FUNCTION_BLOCK CardboardCornerGuardEx
VAR_IN_OUT //controls
	execute : BOOL;
	stop : BOOL;
	
	manualStep : BOOL;
	manualSuction : BOOL;
END_VAR
VAR_IN_OUT
	benderLeft : FoldingMachine;
	
	robotLeft, robotRight : RobotA22;
	
	skidLeft, skidRight : SkidMagazine;
	magazineLeft, magazineRight : SkidMagazine;
	
	wrapper : WrapMachine;
	
	horizontalDriveLeft, horizontalDriveRight : ServoNC;
	verticalDriveLeft, verticalDriveRight : ClearLinkMC;
	pistonBottom : SimplePiston;
	
	suctionTopLeft : ARRAY[*(*1..3*)] OF SuctionPad;
	suctionTopRight : ARRAY[*(*1..3*)] OF SuctionPad;
	suctionBottomLeft : ARRAY[*(*1..3*)] OF SuctionPad; 
	suctionBottomRight : ARRAY[*(*1..3*)] OF SuctionPad;
END_VAR
VAR_OUTPUT
	generalError : BOOL;
	failLeft, failRight : BOOL;
END_VAR
VAR //for testing only
	latchLeft, latchRight : BOOL; //prevents sliders from overshooting the inner limit sensor
	
	suctionEnableTopLeft : BOOL;
	suctionEnableTopRight : BOOL;
	suctionEnableBottomLeft : BOOL;
	suctionEnableBottomRight : BOOL;
	
	ready : BOOL;
	done : BOOL;
END_VAR
VAR	
	step : (IDLE, LOAD_CORNERS, LOAD_FLATS, PUSH, TARGET_WRAP_POSITION, WRAP_AND_RELEASE, COMPLETE := 1050);
	iPair : INT;
	
	masterLoadStep : INT;
	loadSet : INT;
	loadStepLeft, loadStepRight : INT;
	cornerSetLeft, cornerSetRight : INT;
	
	iWrap : INT;
	wrapPoints : INT;
	wrapRotations : INT;
	masterLength : INT;
	
	releaseDelayTimer : TON;
END_VAR
VAR //local types
	topLeftFoldsArr, topRightFoldsArr, bottomLeftFoldsArr, bottomRightFoldsArr : ARRAY[0..GVL.maxPairs] OF INT;
	materialsArr : ARRAY[0..GVL.maxPairs] OF PositionMaterials := [
		(
			position := 0,
			top := 'CAR20M',
			left := 'CAR20S',
			right := 'CAR20S',
			bottom := 'CAR20L',
			topLeft := 'CAR28M',
			topRight := 'CAR28S',
			bottomLeft := 'CAR28S',
			bottomRight := 'CAR28L',
			wrapPoints := 1,
			wrapRotations := 4
		),
		(
			position := 0,
			topLeft := 'COR48',
			topRight := 'COR48',
			bottomLeft := 'COR48',
			bottomRight := 'COR48'
		)];
	
	demoHeight : REAL := 600; //600mm, 60cm
	
	insertionLeft, insertionRight : Insertion;
	innerLoadedMaterials, outerLoadedMaterials : ARRAY[Surface.TOP..Surface.BOTTOM_RIGHT] OF STRING;
	//inner: cardboard by default
	//outer: corner guard by default
END_VAR
VAR CONSTANT
	sectionID : SectionEnum := SectionEnum.CARDBOARD_CORNERGUARD;
	releaseDelay : TIME := T#2000MS;
END_VAR
VAR
	//AOIs encapsulate functionality and reduce the number of module variables
	aoiLoadCornerGuardLeft, aoiLoadCornerGuardRight : AOI_LoadCornerGuard;
	aoiLoadFlatCardboardLeft, aoiLoadFlatCardboardRight : AOI_LoadFlatCardboard;
END_VAR

callLocalModules();

IF stop THEN //may need to turn off suction
	insertionLeft.stop();
	insertionRight.stop();
	pistonBottom.stop();
	
	robotLeft.clearCommand();
	robotRight.clearCommand();
	RETURN;
END_IF

IF NOT (insertionLeft.homingComplete AND insertionRight.homingComplete) THEN
	insertionLeft.homingSequence();
	insertionRight.homingSequence();
	pistonBottom.retract();
END_IF

CASE step OF
	IDLE:
		IF execute THEN
			execute := FALSE;
			step := LOAD_CORNERS;
		END_IF
	
	LOAD_CORNERS:
		IF load(pairIndex := iPair) THEN
			IF manualStep AND_THEN NOT execute THEN
				RETURN;
			END_IF
		
			step := LOAD_FLATS;
		END_IF

	LOAD_FLATS:
		IF loadFlats(pair := materialsArr[iPair]) THEN
			IF manualStep AND_THEN NOT execute THEN
				RETURN;
			END_IF
			
			step := PUSH;
		END_IF
		
	PUSH:
		IF
			NOT insertionLeft.align(1000-demoHeight) OR
			NOT insertionRight.align(1000-demoHeight)
		THEN
			RETURN;
		END_IF
		
		insertionLeft.press();
		insertionRight.press();
		pistonBottom.extend();
		
		IF pistonBottom.extended AND insertionLeft.contact AND insertionRight.contact THEN
			step := TARGET_WRAP_POSITION;
		END_IF
		
	TARGET_WRAP_POSITION:		
		IF iWrap >= wrapPoints THEN
			step := COMPLETE;
			RETURN;
		END_IF
		
		//loadNextPair := materialsArr[iPair].position = materialsArr[iPair + 1].position;	
		
		IF materialsArr[iPair].position = materialsArr[iPair + 1].position THEN
			masterLength := MAX( GetPairMasterLength(materialsArr[iPair]), GetPairMasterLength(materialsArr[iPair + 1]) );
			wrapPoints := MAX( materialsArr[iPair].wrapPoints, materialsArr[iPair + 1].wrapPoints );
			wrapRotations := MAX( materialsArr[iPair].wrapRotations, materialsArr[iPair + 1].wrapRotations );
		ELSE
			masterLength := GetPairMasterLength(materialsArr[iPair]);
			wrapPoints := materialsArr[iPair].wrapPoints;
			wrapRotations := materialsArr[iPair].wrapRotations;
		END_IF
		
		(*
		directionCheckAndSet(
			wrapConveyorPos,
			(currentPair.position - masterLength/2) + (masterLength/(currentPair.wrapPoints + 1) * (iWrap + 1)));
		*)
		step := WRAP_AND_RELEASE;
		
	WRAP_AND_RELEASE:
		releaseDelayTimer(IN:= , PT:= releaseDelay, Q=> , ET=> );
		
		IF wrapper.ready THEN
			wrapper.wrap(wrapRotations);
			releaseDelayTimer.IN := TRUE;
		END_IF
		
		IF releaseDelayTimer.Q THEN
			SetSuctions(suctions := suctionTopLeft, state := FALSE);
			SetSuctions(suctions := suctionTopRight, state := FALSE);
			SetSuctions(suctions := suctionBottomLeft, state := FALSE);
			SetSuctions(suctions := suctionBottomRight, state := FALSE);
			
			insertionLeft.align(0);
			insertionRight.align(0);
			insertionLeft.release();
			insertionRight.release();
			
			pistonBottom.retract();
		END_IF
		
		IF wrapper.done AND insertionLeft.home AND insertionRight.home AND pistonBottom.retracted THEN
			releaseDelayTimer.IN := FALSE;
			step := WRAP_AND_RELEASE;
		END_IF
	
	COMPLETE:
		iPair := (iPair + 1) MOD GVL.maxPairs;
		iWrap := wrapPoints := wrapRotations := 0;
		step := IDLE;
		
END_CASE

ACTION blocks:
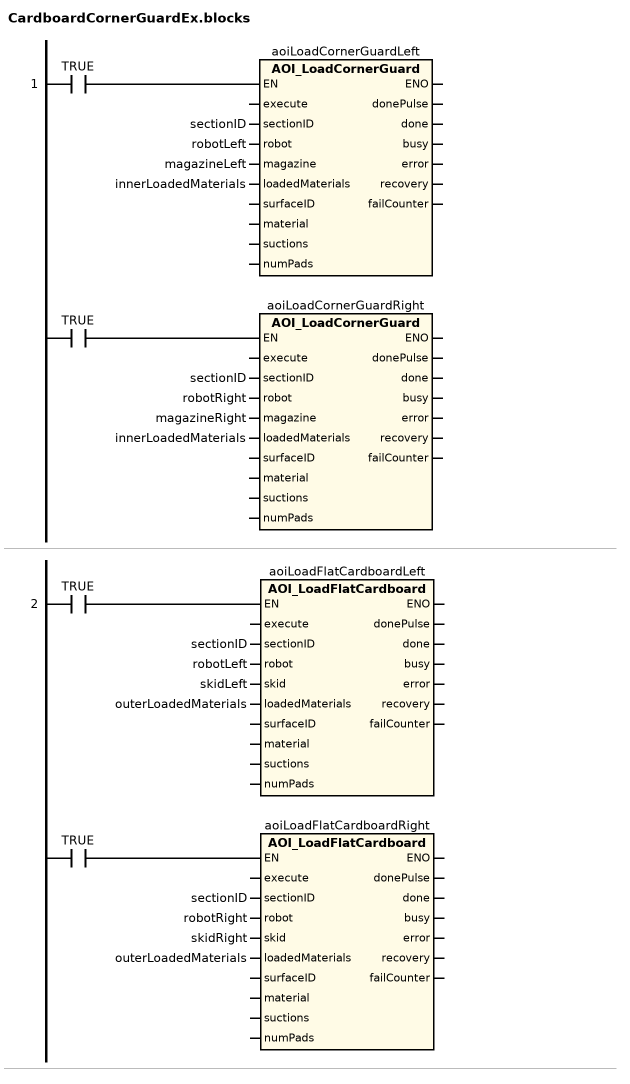
// NETWORK 1
aoiLoadCornerGuardLeft(
    sectionID := sectionID,
    robot := robotLeft,
    magazine := magazineLeft,
    loadedMaterials := innerLoadedMaterials); // AOI_LoadCornerGuard
aoiLoadCornerGuardRight(
    sectionID := sectionID,
    robot := robotRight,
    magazine := magazineRight,
    loadedMaterials := innerLoadedMaterials); // AOI_LoadCornerGuard

// NETWORK 2
aoiLoadFlatCardboardLeft(
    sectionID := sectionID,
    robot := robotLeft,
    skid := skidLeft,
    loadedMaterials := outerLoadedMaterials); // AOI_LoadFlatCardboard
aoiLoadFlatCardboardRight(
    sectionID := sectionID,
    robot := robotRight,
    skid := skidRight,
    loadedMaterials := outerLoadedMaterials); // AOI_LoadFlatCardboard
END_ACTION

ACTION callLocalModules:
{warning disable C0371}
insertionLeft(
	enable:= TRUE, 
	slider:= verticalDriveLeft, 
	screw:= horizontalDriveLeft, 
	contact=> , 
	softContact=> , 
	busy=> , 
	error=> , 
	home=> , 
	homingComplete=> , 
	sliderPos=> );
	
insertionRight(
	enable:= TRUE, 
	slider:= verticalDriveRight, 
	screw:= horizontalDriveRight, 
	contact=> , 
	softContact=> , 
	busy=> , 
	error=> , 
	home=> , 
	homingComplete=> , 
	sliderPos=> );
END_ACTION

METHOD PROTECTED leftCornerSequence : BOOL
VAR_IN_OUT
	robot : RobotA22;
	skid : SkidMagazine;
	suctions : POINTER TO SuctionPad; //ARRAY[*] OF SuctionPad;
	loadStep : INT;
END_VAR
VAR_INPUT
	surfaceID : Surface;
	material : STRING;
	foldPos0 : INT;
	foldPos1 : INT;
END_VAR
VAR_OUTPUT
	error : BOOL;
END_VAR
VAR
	column : INT;
END_VAR
VAR CONSTANT
	suctionDistance : INT := 10;
END_VAR
{warning disable C0371}
IF material = '' THEN
	leftCornerSequence := TRUE;
	RETURN;
END_IF

benderLeft.setFoldingPositions(foldPos0, foldPos1);

CASE loadStep OF
	0:
		robot.clearCommand();
		IF robot.Ready AND overhead = '' THEN
			loadStep := 10;
		END_IF
		
	10: //skid to bender
		IF NOT skid.findSlot(materialID:= material, index=> column) THEN
			error := TRUE;
			RETURN;
		END_IF
		
		(*
		IF robot.eoatDistance < suctionDistance THEN
			robot.HoldMaterial := skid.getSlot(i := column);
		END_IF
		*)
		
		IF robot.Done THEN
			loadStep := 20;
			RETURN;
		END_IF
		
		robot.setGroup(group := 1, value := A22.TRANSFER_TO_BENDER);
		robot.setGroup(group := 2, value := foldPos0);
		robot.setGroup(group := 3, value := foldPos1);
		
	20: //bend
		//IF benderLeft.done THEN
			loadStep := 30;
		//END_IF
		
	30: //bender to overhead or left insertion
		IF wrapper.trayOccupied AND wrapper.Overhead = '' AND robot.HoldMaterial <> '' THEN
			wrapper.Overhead := robot.HoldMaterial;
			robot.HoldMaterial := '';
		END_IF
	
		IF robot.Done THEN
			loadStep := COMPLETE;
			RETURN;
		END_IF
		
		CASE surfaceID OF
			Surface.TOP_RIGHT:		robot.setGroup(group := 1, value := A22.TRANSFER_TO_OVERHEAD);
			Surface.BOTTOM_RIGHT:	robot.setGroup(group := 1, value := A22.TRANSFER_TO_OVERHEAD);
			Surface.TOP_LEFT:		robot.setGroup(group := 1, value := A22.LOAD_BENDER_TO_UPPER_CORNER);
			Surface.BOTTOM_LEFT:	robot.setGroup(group := 1, value := A22.LOAD_BENDER_TO_LOWER_CORNER);
		END_CASE
		robot.setGroup(group := 2, value := 0);
		robot.setGroup(group := 3, value := 0);
	
	COMPLETE:
		CASE surfaceID OF
			Surface.TOP_LEFT:		suctionTopLeft[1].enable := suctionTopLeft[3].enable := TRUE;
			Surface.BOTTOM_LEFT:	suctionBottomLeft[1].enable := suctionBottomLeft[3].enable := TRUE;
		END_CASE
		
		leftCornerSequence := TRUE;
		
END_CASE
END_METHOD

METHOD PROTECTED load : BOOL
VAR_INPUT
	pairIndex : INT;
END_VAR
VAR
	pair : REFERENCE TO PositionMaterials REF= materialsArr[pairIndex];
	nextPair : REFERENCE TO PositionMaterials;
END_VAR
(*
unlike other sections, the load() function for cardboard + corner guard only loads the corners
to load flat cardboards, use the function loadFlats()
*)
{warning disable C0371}

IF robotLeft.error OR robotRight.error THEN
	RETURN;
ELSIF NOT (robotLeft.reserve(sectionID) AND robotRight.reserve(sectionID)) THEN //both robots must be reserved first
	RETURN;
END_IF

IF pairIndex + 1 < GVL.maxPairs THEN
	nextPair REF= materialsArr[pairIndex + 1];
END_IF

CASE masterLoadStep OF
	0: //next pair (which is to be placed over this pair) has the same position as this pair
		IF pairIndex + 1 >= GVL.maxPairs THEN //no next pair
			masterLoadStep := 10;
		ELSIF pair.position < nextPair.position THEN
			masterLoadStep := 10;
		ELSIF MatchesMaterialType(pair:= nextPair, materialType:= 'CAR') AND_THEN loadCornerCardboards(pairIndex:= pairIndex + 1) THEN
			masterLoadStep := 10;
		ELSIF MatchesMaterialType(pair:= nextPair, materialType:= 'COR') AND_THEN loadCornerGuards(pairIndex:= pairIndex + 1) THEN
			masterLoadStep := 10;
		END_IF
		
	10:
		IF
			MatchesMaterialType(pair:= pair, materialType:= 'CAR') AND_THEN loadCornerCardboardsEx(pairIndex:= iPair) OR_ELSE
			MatchesMaterialType(pair:= pair, materialType:= 'COR') AND_THEN loadCornerGuards(pairIndex:= iPair)
		THEN //is cardboard
			masterLoadStep := COMPLETE;
		END_IF
	
	COMPLETE:
		robotLeft.release(sectionID);
		robotRight.release(sectionID);
		
		masterLoadStep := 0;
		load := TRUE;
	
END_CASE
END_METHOD

METHOD PROTECTED loadCornerCardboards : BOOL
VAR_INPUT
	pairIndex : INT;
END_VAR
VAR
	leftSuctionArr, rightSuctionArr : POINTER TO SuctionPad;
	leftNextSet, rightNextSet : INT;
	leftMaterial, rightMaterial : STRING;
	leftFold, rightFold : INT;
	
	pair : REFERENCE TO PositionMaterials REF= materialsArr[pairIndex];
	topLeftFold : INT := topLeftFoldsArr[pairIndex];
	topRightFold : INT := topRightFoldsArr[pairIndex];
	bottomLeftFold : INT := bottomLeftFoldsArr[pairIndex];
	bottomRightFold : INT := bottomRightFoldsArr[pairIndex];
END_VAR
{warning disable C0371}
CASE cornerSetLeft OF
	0:
		leftNextSet := Surface.TOP_RIGHT;
		cornerSetLeft := 0;
		
	Surface.TOP_RIGHT: 
		leftNextSet := Surface.TOP_LEFT;
		leftSuctionArr := suctionTopRight;
		leftMaterial := pair.topRight;
		leftFold := topRightFold;
		
	Surface.TOP_LEFT: 
		leftNextSet := Surface.BOTTOM_RIGHT;
		leftSuctionArr := suctionTopLeft;
		leftMaterial := pair.topLeft;
		leftFold := topLeftFold;
		
	Surface.BOTTOM_RIGHT:
		leftNextSet := Surface.BOTTOM_LEFT;
		leftSuctionArr := suctionBottomRight;
		leftMaterial := pair.bottomRight;
		leftFold := bottomRightFold;
		
	Surface.BOTTOM_LEFT: 
		leftNextSet := COMPLETE;
		leftSuctionArr := suctionBottomLeft;
		leftMaterial := pair.bottomLeft;
		leftFold := bottomLeftFold;
END_CASE
IF
	(cornerSetLeft = 0 OR cornerSetLeft = COMPLETE) OR_ELSE
	leftCornerSequence(
		robot:= robotLeft, 
		skid:= skidLeft, 
		suctions := leftSuctionArr,
		loadStep:= loadStepLeft, 
		surfaceID:= cornerSetLeft,
		material:= pair.topRight, 
		foldPos0:= topRightFold, 
		foldPos1:= 0, 
		error=> )
THEN
	cornerSetLeft := leftNextSet;
	loadStepLeft := 0;
END_IF


CASE cornerSetRight OF
	0:
		cornerSetRight := Surface.TOP_RIGHT;
		rightSuctionArr := suctionTopRight;
		
	Surface.TOP_RIGHT:		
		rightNextSet := Surface.BOTTOM_RIGHT;
		rightSuctionArr := suctionTopRight;
		rightMaterial := pair.topRight;
		rightFold := topRightFold;
		
	Surface.BOTTOM_RIGHT: 
		rightNextSet := COMPLETE;
		rightSuctionArr := suctionBottomRight;
		rightMaterial := pair.bottomRight;
		rightFold := bottomRightFold;		
END_CASE
IF
	(cornerSetRight = 0 OR cornerSetRight = COMPLETE) OR_ELSE
	rightCornerSequence(
		robot:= robotRight, 
		skid:= skidRight, 
		suctions := rightSuctionArr,
		loadStep:= loadStepRight, 
		material:= pair.topRight, 
		surfaceID:= cornerSetRight,
		foldPos0:= pair.topRightFold, 
		foldPos1:= 0, 
		error=> )
THEN
	cornerSetRight := rightNextSet;
	loadStepRight := 0;
END_IF



IF cornerSetLeft = COMPLETE AND cornerSetRight = COMPLETE THEN
	loadCornerCardboards := TRUE;
	
	loadStepLeft := loadStepRight := 0;
	cornerSetLeft := cornerSetRight := 0;
END_IF
END_METHOD

METHOD PROTECTED loadCornerCardboardsEx : BOOL
VAR_INPUT
	pairIndex : INT;
END_VAR
VAR
	suctionsArrLeft, suctionsArrRight : POINTER TO SuctionPad;
	nextSetLeft, nextSetRight : INT;

	pair : REFERENCE TO PositionMaterials REF= materialsArr[pairIndex];
	topLeftFold : INT := topLeftFoldsArr[pairIndex];
	topRightFold : INT := topRightFoldsArr[pairIndex];
	bottomLeftFold : INT := bottomLeftFoldsArr[pairIndex];
	bottomRightFold : INT := bottomRightFoldsArr[pairIndex];
END_VAR
{warning disable C0371}
CASE cornerSetLeft OF
	0:
		cornerSetLeft := Surface.TOP_RIGHT;
		loadStepLeft := 0;
		
	Surface.TOP_RIGHT: 
		IF
			leftCornerSequence(
				robot:= robotLeft, 
				skid:= skidLeft, 
				suctions := suctionTopRight,
				loadStep:= loadStepLeft, 
				surfaceID:= Surface.TOP_RIGHT,
				material:= pair.topRight, 
				foldPos0:= topRightFold, 
				foldPos1:= 0, 
				error=> )
		THEN
			cornerSetLeft := Surface.TOP_LEFT;
			loadStepLeft := 0;
		END_IF
		
	Surface.TOP_LEFT: 
		IF
			leftCornerSequence(
				robot:= robotLeft, 
				skid:= skidLeft, 
				suctions := suctionTopLeft,
				loadStep:= loadStepLeft, 
				surfaceID:= Surface.TOP_LEFT,
				material:= pair.topLeft, 
				foldPos0:= topLeftFold, 
				foldPos1:= 0, 
				error=> )
		THEN
			cornerSetLeft := Surface.BOTTOM_RIGHT;
			loadStepLeft := 0;
		END_IF
		
	Surface.BOTTOM_RIGHT: 
		IF
			leftCornerSequence(
				robot:= robotLeft, 
				skid:= skidLeft, 
				suctions := suctionBottomRight,
				loadStep:= loadStepLeft, 
				surfaceID:= Surface.BOTTOM_RIGHT,
				material:= pair.bottomRight, 
				foldPos0:= bottomRightFold, 
				foldPos1:= 0, 
				error=> )
		THEN
			cornerSetLeft := Surface.BOTTOM_LEFT;
			loadStepLeft := 0;
		END_IF
		
	Surface.BOTTOM_LEFT: 
		IF
			leftCornerSequence(
				robot:= robotLeft, 
				skid:= skidLeft, 
				suctions := suctionBottomLeft,
				loadStep:= loadStepLeft, 
				surfaceID:= Surface.BOTTOM_LEFT,
				material:= pair.bottomLeft, 
				foldPos0:= bottomLeftFold, 
				foldPos1:= 0, 
				error=> )
		THEN
			cornerSetLeft := COMPLETE;
			loadStepLeft := 0;
		END_IF
END_CASE

//------------------------------------------------------------
CASE cornerSetRight OF
	0:
		cornerSetRight := Surface.TOP_RIGHT;
		loadStepRight := 0;
		
	Surface.TOP_RIGHT: 
		IF
			rightCornerSequence(
				robot:= robotRight, 
				skid:= skidRight, 
				suctions := suctionTopRight,
				loadStep:= loadStepRight, 
				surfaceID:= Surface.TOP_RIGHT,
				material:= pair.topRight, 
				foldPos0:= topRightFold, 
				foldPos1:= 0, 
				error=> )
		THEN
			cornerSetRight := Surface.BOTTOM_RIGHT;
			loadStepRight := 0;
		END_IF
		
	Surface.BOTTOM_RIGHT: 
		IF
			rightCornerSequence(
				robot:= robotRight, 
				skid:= skidRight, 
				suctions := suctionBottomRight,
				loadStep:= loadStepRight, 
				surfaceID:= Surface.BOTTOM_RIGHT,
				material:= pair.bottomRight, 
				foldPos0:= bottomRightFold, 
				foldPos1:= 0, 
				error=> )
		THEN
			cornerSetRight := Surface.BOTTOM_RIGHT;
			loadStepRight := 0;
		END_IF
		
		cornerSetRight := COMPLETE;			
		loadStepRight := COMPLETE;
		
END_CASE

//------------------------------------------------------------
IF cornerSetLeft = COMPLETE AND cornerSetRight = COMPLETE THEN
	loadCornerCardboardsEx := TRUE;
	
	loadStepLeft := loadStepRight := 0;
	cornerSetLeft := cornerSetRight := 0;
END_IF
END_METHOD

METHOD PROTECTED loadCornerGuards : BOOL
VAR_INPUT
	pairIndex : INT;
END_VAR
VAR_OUTPUT
	fail : BOOL;
END_VAR
VAR
	pair : REFERENCE TO PositionMaterials REF= materialsArr[pairIndex];
END_VAR
{warning disable C0371}
CASE loadSet OF
	0: //upper corners
		IF 
			loadGuardSequence(
				robot:= robotLeft, 
				magazine:= magazineLeft, 
				suctions:= suctionTopLeft,
				loadStep:= loadStepLeft, 
				surfaceID:= Surface.TOP_LEFT, 
				material:= pair.topLeft, 
				error=> failLeft)
			AND
			loadGuardSequence(
				robot:= robotRight, 
				magazine:= magazineLeft,
				suctions:= suctionTopRight,
				loadStep:= loadStepRight, 
				surfaceID:= Surface.TOP_RIGHT, 
				material:= pair.topRight, 
				error=> failRight)
		THEN
			loadStepLeft := loadStepRight := 0;
			loadSet := 10;
		END_IF
		
	10: //lower corners
		IF 
			loadGuardSequence(
				robot:= robotLeft, 
				magazine:= skidLeft, 
				suctions:= suctionTopLeft,
				loadStep:= loadStepLeft, 
				surfaceID:= Surface.BOTTOM_LEFT, 
				material:= pair.bottomLeft, 
				error=> failLeft)
			AND
			loadGuardSequence(
				robot:= robotRight, 
				magazine:= skidRight,
				suctions:= suctionTopRight,
				loadStep:= loadStepRight, 
				surfaceID:= Surface.BOTTOM_RIGHT, 
				material:= pair.bottomRight, 
				error=> failRight)
		THEN
			loadStepLeft := loadStepRight := 0;
			loadSet := COMPLETE;
		END_IF
	
	COMPLETE:
		loadStepLeft := loadStepRight := 0;
		loadSet := 0;
		
		loadCornerGuards := TRUE;
END_CASE

fail := failLeft OR failRight;
END_METHOD

METHOD PROTECTED loadFlats : BOOL
VAR_INPUT
	pair : REFERENCE TO PositionMaterials;
END_VAR
VAR_OUTPUT
	error : BOOL;
END_VAR
{warning disable C0371}
CASE loadSet OF
	0: //top and bottom
		IF 
			loadFlatSequence(
				robot:= robotLeft, 
				skid:= skidLeft, 
				loadStep:= loadStepLeft, 
				surfaceID:= Surface.TOP, 
				material:= pair.top, 
				fail=> )
			AND
			loadFlatSequence(
				robot:= robotRight, 
				skid:= skidRight, 
				loadStep:= loadStepRight, 
				surfaceID:= Surface.BOTTOM, 
				material:= pair.bottom, 
				fail=> )
		THEN
			loadStepLeft := loadStepRight := 0;
			loadSet := 10;
		END_IF
		
	10: //sides
		IF 
			loadFlatSequence(
				robot:= robotLeft, 
				skid:= skidLeft, 
				loadStep:= loadStepLeft, 
				surfaceID:= Surface.LEFT, 
				material:= pair.left, 
				fail=> )
			AND
			loadFlatSequence(
				robot:= robotRight, 
				skid:= skidRight, 
				loadStep:= loadStepRight, 
				surfaceID:= Surface.RIGHT, 
				material:= pair.right, 
				fail=> )
		THEN
			loadStepLeft := loadStepRight := 0;
			loadSet := COMPLETE;
		END_IF
	
	COMPLETE:
		loadStepLeft := loadStepRight := 0;
		loadSet := 0;
		
		loadFlats := TRUE;
END_CASE
END_METHOD

METHOD loadFlatSequence : BOOL
VAR_IN_OUT
	robot : RobotA22;
	skid : SkidMagazine;
	loadStep : INT;
END_VAR
VAR_INPUT
	surfaceID : Surface;
	material : STRING;
END_VAR
VAR_OUTPUT
	fail : BOOL;
END_VAR
VAR
	task : INT;
	slot : INT;
END_VAR
IF material = '' THEN
	loadFlatSequence := TRUE;
	RETURN;
END_IF

CASE loadStep OF
	0:
		robot.clearCommand();
		IF robot.Ready THEN
			step := 10;
		END_IF
		
	10: //storage to gripper
		IF NOT skid.findSlot(materialID := material, index => slot) THEN
			fail := TRUE;
			RETURN;
		END_IF
		
		IF robot.Done THEN
			loadStep := COMPLETE;
			RETURN;
		END_IF
		
		CASE surfaceID OF
			Surface.TOP: 					task := A22.LOAD_CARDBOARD_TOP;
			Surface.LEFT, Surface.RIGHT: 	task := A22.LOAD_CARDBOARD_SIDE;
			Surface.BOTTOM: 				task := A22.LOAD_CARDBOARD_BOTTOM;
		END_CASE
		
		robot.setGroup(group := 1, value := task);
		robot.setGroup(group := 2, value := slot);
		
	20: //gripper to insertion
		
	COMPLETE:
		loadFlatSequence := TRUE;
	
END_CASE
END_METHOD

METHOD loadGuardSequence : BOOL
VAR_IN_OUT
	robot : RobotA22;
	magazine : SkidMagazine;
	suctions : ARRAY[*] OF SuctionPad;
	loadStep : INT;
END_VAR
VAR_INPUT
	surfaceID : Surface;
	material : STRING;
END_VAR
VAR_OUTPUT
	error : BOOL;
END_VAR
VAR
	task : INT;
	slot : INT;
END_VAR
IF material = '' THEN
	loadGuardSequence := TRUE;
	RETURN;
END_IF

CASE loadStep OF
	0:
		IF NOT magazine.findSlot(materialID := material, index => slot) THEN //load from staging table
			error := TRUE;
			RETURN;
		END_IF
		
		IF robot.Done THEN
			loadStep := COMPLETE;
			RETURN;
		END_IF
		
		CASE surfaceID OF
			Surface.TOP_LEFT, Surface.TOP_RIGHT: 		task := A22.LOAD_CORNER_GUARD_UPPER;
			Surface.BOTTOM_LEFT, Surface.BOTTOM_RIGHT:	task := A22.LOAD_CORNER_GUARD_LOWER;
		END_CASE
		
		robot.setGroup(group := 1, value := task);
		robot.setGroup(group := 2, value := slot);
		
	COMPLETE:
		suctions[2].enable := TRUE;
		loadGuardSequence := TRUE;
END_CASE
END_METHOD

METHOD PROTECTED loadLeftCornerCardboards : BOOL
VAR_INPUT
	pair : REFERENCE TO PositionMaterials;
END_VAR
VAR
	suctionsArrLeft, suctionsArrRight : POINTER TO SuctionPad;
	nextSetLeft, nextSetRight : INT;
END_VAR
{warning disable C0371}
CASE cornerSetLeft OF
	0:
		cornerSetLeft := Surface.TOP_RIGHT;
		loadStepLeft := 0;
		
	Surface.TOP_RIGHT: 
		IF
			leftCornerSequence(
				robot:= robotLeft, 
				skid:= skidLeft, 
				suctions := suctionTopRight,
				loadStep:= loadStepLeft, 
				surfaceID:= Surface.TOP_RIGHT,
				material:= pair.topRight, 
				foldPos0:= pair.topRightFold, 
				foldPos1:= 0, 
				error=> )
		THEN
			cornerSetLeft := Surface.TOP_LEFT;
			loadStepLeft := 0;
		END_IF
		
	Surface.TOP_LEFT: 
		IF
			leftCornerSequence(
				robot:= robotLeft, 
				skid:= skidLeft, 
				suctions := suctionTopLeft,
				loadStep:= loadStepLeft, 
				surfaceID:= Surface.TOP_LEFT,
				material:= pair.topLeft, 
				foldPos0:= pair.topLeftFold, 
				foldPos1:= 0, 
				error=> )
		THEN
			cornerSetLeft := Surface.BOTTOM_RIGHT;
			loadStepLeft := 0;
		END_IF
		
	Surface.BOTTOM_RIGHT: 
		IF
			leftCornerSequence(
				robot:= robotLeft, 
				skid:= skidLeft, 
				suctions := suctionBottomRight,
				loadStep:= loadStepLeft, 
				surfaceID:= Surface.BOTTOM_RIGHT,
				material:= pair.bottomRight, 
				foldPos0:= pair.bottomRightFold, 
				foldPos1:= 0, 
				error=> )
		THEN
			cornerSetLeft := Surface.BOTTOM_LEFT;
			loadStepLeft := 0;
		END_IF
		
	Surface.BOTTOM_LEFT: 
		IF
			leftCornerSequence(
				robot:= robotLeft, 
				skid:= skidLeft, 
				suctions := suctionBottomLeft,
				loadStep:= loadStepLeft, 
				surfaceID:= Surface.BOTTOM_LEFT,
				material:= pair.bottomLeft, 
				foldPos0:= pair.bottomLeftFold, 
				foldPos1:= 0, 
				error=> )
		THEN
			cornerSetLeft := COMPLETE;
			loadStepLeft := 0;
		END_IF
END_CASE

//------------------------------------------------------------
IF cornerSetLeft = COMPLETE THEN
	loadStepLeft := 0;
	cornerSetLeft := 0;
	loadLeftCornerCardboards := TRUE;
END_IF
END_METHOD

METHOD PROTECTED loadRightCornerCardboards : BOOL
VAR_INPUT
	pair : REFERENCE TO PositionMaterials;
END_VAR
VAR
	suctionsArrLeft, suctionsArrRight : POINTER TO SuctionPad;
	nextSetLeft, nextSetRight : INT;
END_VAR
{warning disable C0371}
CASE cornerSetRight OF
	0:
		cornerSetRight := Surface.TOP_RIGHT;
		loadStepRight := 0;
		
	Surface.TOP_RIGHT: 
		IF
			rightCornerSequence(
				robot:= robotRight, 
				skid:= skidRight, 
				suctions := suctionTopRight,
				loadStep:= loadStepRight, 
				surfaceID:= Surface.TOP_RIGHT,
				material:= pair.topRight, 
				foldPos0:= pair.topRightFold, 
				foldPos1:= 0, 
				error=> )
		THEN
			cornerSetRight := Surface.BOTTOM_RIGHT;
			loadStepRight := 0;
		END_IF
		
	Surface.BOTTOM_RIGHT: 
		IF
			rightCornerSequence(
				robot:= robotRight, 
				skid:= skidRight, 
				suctions := suctionBottomRight,
				loadStep:= loadStepRight, 
				surfaceID:= Surface.BOTTOM_RIGHT,
				material:= pair.bottomRight, 
				foldPos0:= pair.bottomRightFold, 
				foldPos1:= 0, 
				error=> )
		THEN
			cornerSetRight := Surface.BOTTOM_RIGHT;
			loadStepRight := 0;
		END_IF
		
		cornerSetRight := COMPLETE;			
		loadStepRight := COMPLETE;
		
END_CASE

//------------------------------------------------------------
IF cornerSetRight = COMPLETE THEN	
	loadStepRight := 0;
	cornerSetRight := 0;
	loadRightCornerCardboards := TRUE;
END_IF
END_METHOD

METHOD PROTECTED rightCornerSequence : BOOL
VAR_IN_OUT
	robot : RobotA22;
	skid : SkidMagazine;
	suctions : POINTER TO SuctionPad; //array of SuctionPads, casts from [1..3] to [0..2]
	loadStep : INT;
END_VAR
VAR_INPUT
	surfaceID : Surface;
	material : STRING;
	foldPos0 : INT;
	foldPos1 : INT;
END_VAR
VAR_OUTPUT
	error : BOOL;
END_VAR
VAR
	column : INT;
END_VAR
VAR CONSTANT
	suctionDistance : INT := 10;
END_VAR
{warning disable C0371}
IF material = '' THEN
	rightCornerSequence := TRUE;
	RETURN;
END_IF

CASE loadStep OF
	0:
		robot.clearCommand();
		IF robot.Ready THEN
			loadStep := 10;
		END_IF
		
	10: //overhead to insertion
		IF wrapper.Overhead = '' THEN
			RETURN;
		END_IF
		(*
		IF robot.eoatDistance < suctionDistance THEN
			robot.HoldMaterial := wrapper.Overhead;
		END_IF
		*)
	
		IF robot.Done THEN
			loadStep := COMPLETE;
			RETURN;
		END_IF
		
		CASE surfaceID OF
			Surface.TOP_RIGHT:		robot.setGroup(group := 1, value := A22.LOAD_OVERHEAD_TO_UPPER_CORNER);
			Surface.BOTTOM_RIGHT:	robot.setGroup(group := 1, value := A22.LOAD_OVERHEAD_TO_LOWER_CORNER);
		END_CASE
		robot.setGroup(group := 2, value := foldPos0);
		robot.setGroup(group := 3, value := foldPos1);
	
	COMPLETE:
		robot.clearCommand();
		
		CASE surfaceID OF
			Surface.TOP_RIGHT:		suctionTopRight[1].enable := suctionTopRight[3].enable := TRUE;
			Surface.BOTTOM_RIGHT:	suctionBottomRight[1].enable := suctionBottomRight[3].enable := TRUE;
		END_CASE
		
		//suctions[0].enable := TRUE;
		//suctions[2].enable := TRUE;
		
		rightCornerSequence := TRUE;
	
END_CASE
END_METHOD

END_FUNCTION_BLOCK

(* stored: Version 1.1.0.1, ProductVersion 3.1.4024.11
   POU CardboardCornerGuardEx: Id {43a9c6e1-e77d-41f5-aea3-07b47a57c140}, SpecialFunc None
   Folder Actions: Id {c8c39f76-dbed-4e64-98b8-9f897e55ef48}
   Folder Cardboard (Corner): Id {75e45005-57b6-45af-977a-1cc75cf19289}
   Folder Cardboard (Flat): Id {69bbbb84-f428-46bc-8482-36bd2217074a}
   Folder Corner Guards: Id {6138b1d4-74c6-4a8f-864e-6193654c592a}
   Folder x_Obsolete: Id {ae97f731-8159-458d-a4c2-1a1c4ac5d0d1}
   Action blocks: Id {42a09ab4-5795-4272-b1bf-07353ead9a10}
   Action callLocalModules: Id {39933dae-94a6-4c04-af7d-ba6ce828a93a}
   Method leftCornerSequence: Id {08bffef9-e349-4b7d-9ae3-92f5a7d8876a}
   Method load: Id {a681c93d-e590-4020-9185-d7ae010cf638}
   Method loadCornerCardboards: Id {fc6e26f1-7233-42c4-a94a-66d2e256266a}
   Method loadCornerCardboardsEx: Id {156f628d-7b56-4840-9717-9971eeb42365}
   Method loadCornerGuards: Id {73216583-3bb4-409e-896a-e96f29db7009}
   Method loadFlats: Id {b9a93d4c-938b-4af6-a5a3-5141d50c48d4}
   Method loadFlatSequence: Id {e9b25173-0158-437d-9616-4153dd5d3500}
   Method loadGuardSequence: Id {6d84fe42-26e5-4a1f-b580-8cefdfabe586}
   Method loadLeftCornerCardboards: Id {5220eb17-3d60-4a35-a2d9-12b1f5a6525f}
   Method loadRightCornerCardboards: Id {ccdab2eb-d382-4ec7-bb9d-d70515ff692c}
   Method rightCornerSequence: Id {879cd7f3-c4e8-4979-a4c5-8a1bacb14790} *)
